FUNCTION_BLOCK Meca500_SetGripperVel
VAR
    Output_Params : array[1..6] of real;
    FirstScan : BOOL := False;
END_VAR
VAR_INPUT
    Execute : BOOL;
    Speed : REAL;
END_VAR
VAR_OUTPUT
    Sent : BOOL;
    Buffered : BOOL;
    Error : BOOL;
END_VAR
VAR_IN_OUT
    Robot : Meca500;
END_VAR
VAR_INPUT
    ExternalStateControl : BOOL;
    ExternalMoveID : UINT;
END_VAR
IF Execute THEN	
	(*Collect Inputs and store them locally*)
	Output_Params[1]:=Speed;
	Output_Params[2]:=0;
	Output_Params[3]:=0;
	Output_Params[4]:=0;
	Output_Params[5]:=0;
	Output_Params[6]:=0;

	(* If Values have change, Reinitialise Outputs*)

	IF FirstScan=0 OR 
		Robot.Outputs.MotionCommand.MoveSubIndex001 <> Output_Params[1] OR 
		Robot.Outputs.MotionCommand.MoveSubIndex002 <> Output_Params[2] OR 
		Robot.Outputs.MotionCommand.MoveSubIndex003 <> Output_Params[3] OR
		Robot.Outputs.MotionCommand.MoveSubIndex004 <> Output_Params[4] OR 
		Robot.Outputs.MotionCommand.MoveSubIndex005 <> Output_Params[5] OR 
		Robot.Outputs.MotionCommand.MoveSubIndex006 <> Output_Params[6] 
	THEN
		Buffered := FALSE;
		Sent := FALSE;
	END_IF;


	(*if not in legacy mode, Act Setpoint*)
	IF Robot.Outputs.MotionControl.MoveID <> 0 THEN
	    Robot.Outputs.MotionControl.SetPoint := TRUE;
	END_IF;

	(* To send _Move, send _Move ID *)
	IF NOT Buffered AND NOT Sent THEN
	    
	    Robot.Outputs.MotionCommand.MoveCommand	:= EnumToNum(Meca500Cmd#SetGripperVel);
	    Robot.Outputs.MotionCommand.MoveSubIndex001 := Output_Params[1];
		Robot.Outputs.MotionCommand.MoveSubIndex002 := Output_Params[2];
		Robot.Outputs.MotionCommand.MoveSubIndex003 := Output_Params[3];
		Robot.Outputs.MotionCommand.MoveSubIndex004 := Output_Params[4];
		Robot.Outputs.MotionCommand.MoveSubIndex005 := Output_Params[5];
		Robot.Outputs.MotionCommand.MoveSubIndex006 := Output_Params[6];
	    
	    IF ExternalStateControl THEN
	        IF ExternalMoveID <> 0 AND ExternalMoveID <> 32190 AND ExternalMoveID <> 32191 THEN
	            Robot.Outputs.MotionControl.MoveID := ExternalMoveID;
	            Sent := TRUE;
	        END_IF;
	        
	    ELSE (*Not External Control*)
	        IF Robot.Outputs.MotionControl.MoveID = 32190 THEN
	            Robot.Outputs.MotionControl.MoveID := 32191;
	        ELSIF Robot.Outputs.MotionControl.MoveID = 32191 THEN
	            Robot.Outputs.MotionControl.MoveID := 32190;
	        ELSIF Robot.Outputs.MotionControl.MoveID <> 32190 OR Robot.Outputs.MotionControl.MoveID <> 32191 THEN
	            Robot.Outputs.MotionControl.MoveID := 32190;
	        END_IF;
	        Sent := TRUE;
	    END_IF;
	END_IF;

	(* Check if command has been sent, if so, check if it was received *)
	IF Sent AND
	    Robot.Outputs.MotionCommand.MoveCommand = EnumToNum(Meca500Cmd#SetGripperVel) AND
	    Robot.Outputs.MotionCommand.MoveSubIndex001 = Output_Params[1] AND 
		Robot.Outputs.MotionCommand.MoveSubIndex002 = Output_Params[2] AND 
		Robot.Outputs.MotionCommand.MoveSubIndex003 = Output_Params[3] AND 
		Robot.Outputs.MotionCommand.MoveSubIndex004 = Output_Params[4] AND 
		Robot.Outputs.MotionCommand.MoveSubIndex005 = Output_Params[5] AND 
		Robot.Outputs.MotionCommand.MoveSubIndex006 = Output_Params[6] AND
		Robot.Inputs.Motion.MoveID = Robot.Outputs.MotionControl.MoveID 
	THEN
		 Buffered := TRUE;
	END_IF;


	(*If External _Move ID is equal to Internal, raise an error*)
	IF ExternalMoveID = 32190 OR ExternalMoveID = 32191 THEN
	    Error := TRUE;
	END_IF;

	FirstScan := TRUE;
ELSE
	FirstScan := False;
	Sent := FALSE;
	Buffered := FALSE;
END_IF;
END_FUNCTION_BLOCK

FUNCTION_BLOCK Meca500_SetJointsAcc
VAR
    Output_Params : array[1..6] of real;
    FirstScan : BOOL := False;
END_VAR
VAR_INPUT
    Execute : BOOL;
    Acceleration_Percentage : REAL;
END_VAR
VAR_OUTPUT
    Sent : BOOL;
    Buffered : BOOL;
    Error : BOOL;
END_VAR
VAR_IN_OUT
    Robot : Meca500;
END_VAR
VAR_INPUT
    ExternalStateControl : BOOL;
    ExternalMoveID : UINT;
END_VAR
IF Execute THEN	
	(*Collect Inputs and store them locally*)
	Output_Params[1]:=Acceleration_Percentage;
	Output_Params[2]:=0;
	Output_Params[3]:=0;
	Output_Params[4]:=0;
	Output_Params[5]:=0;
	Output_Params[6]:=0;

	(* If Values have change, Reinitialise Outputs*)

	IF FirstScan=0 OR 
		Robot.Outputs.MotionCommand.MoveSubIndex001 <> Output_Params[1] OR 
		Robot.Outputs.MotionCommand.MoveSubIndex002 <> Output_Params[2] OR 
		Robot.Outputs.MotionCommand.MoveSubIndex003 <> Output_Params[3] OR
		Robot.Outputs.MotionCommand.MoveSubIndex004 <> Output_Params[4] OR 
		Robot.Outputs.MotionCommand.MoveSubIndex005 <> Output_Params[5] OR 
		Robot.Outputs.MotionCommand.MoveSubIndex006 <> Output_Params[6] 
	THEN
		Buffered := FALSE;
		Sent := FALSE;
	END_IF;


	(*if not in legacy mode, Act Setpoint*)
	IF Robot.Outputs.MotionControl.MoveID <> 0 THEN
	    Robot.Outputs.MotionControl.SetPoint := TRUE;
	END_IF;

	(* To send _Move, send _Move ID *)
	IF NOT Buffered AND NOT Sent THEN
	    
	    Robot.Outputs.MotionCommand.MoveCommand	:= EnumToNum(Meca500Cmd#SetJointAcc);
	    Robot.Outputs.MotionCommand.MoveSubIndex001 := Output_Params[1];
		Robot.Outputs.MotionCommand.MoveSubIndex002 := Output_Params[2];
		Robot.Outputs.MotionCommand.MoveSubIndex003 := Output_Params[3];
		Robot.Outputs.MotionCommand.MoveSubIndex004 := Output_Params[4];
		Robot.Outputs.MotionCommand.MoveSubIndex005 := Output_Params[5];
		Robot.Outputs.MotionCommand.MoveSubIndex006 := Output_Params[6];
	    
	    IF ExternalStateControl THEN
	        IF ExternalMoveID <> 0 AND ExternalMoveID <> 32090 AND ExternalMoveID <> 32091 THEN
	            Robot.Outputs.MotionControl.MoveID := ExternalMoveID;
	            Sent := TRUE;
	        END_IF;
	        
	    ELSE (*Not External Control*)
	        IF Robot.Outputs.MotionControl.MoveID = 32090 THEN
	            Robot.Outputs.MotionControl.MoveID := 32091;
	        ELSIF Robot.Outputs.MotionControl.MoveID = 32091 THEN
	            Robot.Outputs.MotionControl.MoveID := 32090;
	        ELSIF Robot.Outputs.MotionControl.MoveID <> 32090 OR Robot.Outputs.MotionControl.MoveID <> 32091 THEN
	            Robot.Outputs.MotionControl.MoveID := 32090;
	        END_IF;
	        Sent := TRUE;
	    END_IF;
	END_IF;

	(* Check if command has been sent, if so, check if it was received *)
	IF Sent AND
	    Robot.Outputs.MotionCommand.MoveCommand = EnumToNum(Meca500Cmd#SetJointAcc) AND
	    Robot.Outputs.MotionCommand.MoveSubIndex001 = Output_Params[1] AND 
		Robot.Outputs.MotionCommand.MoveSubIndex002 = Output_Params[2] AND 
		Robot.Outputs.MotionCommand.MoveSubIndex003 = Output_Params[3] AND 
		Robot.Outputs.MotionCommand.MoveSubIndex004 = Output_Params[4] AND 
		Robot.Outputs.MotionCommand.MoveSubIndex005 = Output_Params[5] AND 
		Robot.Outputs.MotionCommand.MoveSubIndex006 = Output_Params[6] AND
		Robot.Inputs.Motion.MoveID = Robot.Outputs.MotionControl.MoveID 
	THEN
		 Buffered := TRUE;
	END_IF;


	(*If External _Move ID is equal to Internal, raise an error*)
	IF ExternalMoveID = 32090 OR ExternalMoveID = 32091 THEN
	    Error := TRUE;
	END_IF;

	FirstScan := TRUE;
ELSE
	FirstScan := False;
	Sent := FALSE;
	Buffered := FALSE;
END_IF;
END_FUNCTION_BLOCK

FUNCTION_BLOCK Meca500_SetJointsVel
VAR
    Output_Params : array[1..6] of real;
    FirstScan : BOOL := False;
END_VAR
VAR_INPUT
    Execute : BOOL;
    Velocity_Percentage : REAL;
END_VAR
VAR_OUTPUT
    Sent : BOOL;
    Buffered : BOOL;
    Error : BOOL;
END_VAR
VAR_IN_OUT
    Robot : Meca500;
END_VAR
VAR_INPUT
    ExternalStateControl : BOOL;
    ExternalMoveID : UINT;
END_VAR
IF Execute THEN	
	(*Collect Inputs and store them locally*)
	Output_Params[1]:=Velocity_Percentage;
	Output_Params[2]:=0;
	Output_Params[3]:=0;
	Output_Params[4]:=0;
	Output_Params[5]:=0;
	Output_Params[6]:=0;

	(* If Values have change, Reinitialise Outputs*)

	IF FirstScan=0 OR 
		Robot.Outputs.MotionCommand.MoveSubIndex001 <> Output_Params[1] OR 
		Robot.Outputs.MotionCommand.MoveSubIndex002 <> Output_Params[2] OR 
		Robot.Outputs.MotionCommand.MoveSubIndex003 <> Output_Params[3] OR
		Robot.Outputs.MotionCommand.MoveSubIndex004 <> Output_Params[4] OR 
		Robot.Outputs.MotionCommand.MoveSubIndex005 <> Output_Params[5] OR 
		Robot.Outputs.MotionCommand.MoveSubIndex006 <> Output_Params[6] 
	THEN
		Buffered := FALSE;
		Sent := FALSE;
	END_IF;


	(*if not in legacy mode, Act Setpoint*)
	IF Robot.Outputs.MotionControl.MoveID <> 0 THEN
	    Robot.Outputs.MotionControl.SetPoint := TRUE;
	END_IF;

	(* To send _Move, send _Move ID *)
	IF NOT Buffered AND NOT Sent THEN
	    
	    Robot.Outputs.MotionCommand.MoveCommand	:= EnumToNum(Meca500Cmd#SetJointVel);
	    Robot.Outputs.MotionCommand.MoveSubIndex001 := Output_Params[1];
		Robot.Outputs.MotionCommand.MoveSubIndex002 := Output_Params[2];
		Robot.Outputs.MotionCommand.MoveSubIndex003 := Output_Params[3];
		Robot.Outputs.MotionCommand.MoveSubIndex004 := Output_Params[4];
		Robot.Outputs.MotionCommand.MoveSubIndex005 := Output_Params[5];
		Robot.Outputs.MotionCommand.MoveSubIndex006 := Output_Params[6];
	    
	    IF ExternalStateControl THEN
	        IF ExternalMoveID <> 0 AND ExternalMoveID <> 32080 AND ExternalMoveID <> 32081 THEN
	            Robot.Outputs.MotionControl.MoveID := ExternalMoveID;
	            Sent := TRUE;
	        END_IF;
	        
	    ELSE (*Not External Control*)
	        IF Robot.Outputs.MotionControl.MoveID = 32080 THEN
	            Robot.Outputs.MotionControl.MoveID := 32081;
	        ELSIF Robot.Outputs.MotionControl.MoveID = 32081 THEN
	            Robot.Outputs.MotionControl.MoveID := 32080;
	        ELSIF Robot.Outputs.MotionControl.MoveID <> 32080 OR Robot.Outputs.MotionControl.MoveID <> 32081 THEN
	            Robot.Outputs.MotionControl.MoveID := 32080;
	        END_IF;
	        Sent := TRUE;
	    END_IF;
	END_IF;

	(* Check if command has been sent, if so, check if it was received *)
	IF Sent AND
	    Robot.Outputs.MotionCommand.MoveCommand = EnumToNum(Meca500Cmd#SetJointVel) AND
	    Robot.Outputs.MotionCommand.MoveSubIndex001 = Output_Params[1] AND 
		Robot.Outputs.MotionCommand.MoveSubIndex002 = Output_Params[2] AND 
		Robot.Outputs.MotionCommand.MoveSubIndex003 = Output_Params[3] AND 
		Robot.Outputs.MotionCommand.MoveSubIndex004 = Output_Params[4] AND 
		Robot.Outputs.MotionCommand.MoveSubIndex005 = Output_Params[5] AND 
		Robot.Outputs.MotionCommand.MoveSubIndex006 = Output_Params[6] AND
		Robot.Inputs.Motion.MoveID = Robot.Outputs.MotionControl.MoveID 
	THEN
		 Buffered := TRUE;
	END_IF;


	(*If External _Move ID is equal to Internal, raise an error*)
	IF ExternalMoveID = 32080 OR ExternalMoveID = 32081 THEN
	    Error := TRUE;
	END_IF;

	FirstScan := TRUE;
ELSE
	FirstScan := False;
	Sent := FALSE;
	Buffered := FALSE;
END_IF;
END_FUNCTION_BLOCK

FUNCTION_BLOCK Meca500_SetTorqueLimitCfg
VAR
    Output_Params : array[1..6] of real;
    FirstScan : BOOL := False;
END_VAR
VAR_INPUT
    Execute : BOOL;
    Severity : REAL;
    Mode : REAL;
END_VAR
VAR_OUTPUT
    Sent : BOOL;
    Buffered : BOOL;
    Error : BOOL;
END_VAR
VAR_IN_OUT
    Robot : Meca500;
END_VAR
VAR_INPUT
    ExternalStateControl : BOOL;
    ExternalMoveID : UINT;
END_VAR
IF Execute THEN	
	(*Collect Inputs and store them locally*)
	Output_Params[1]:=Severity;
	Output_Params[2]:=Mode;
	Output_Params[3]:=0;
	Output_Params[4]:=0;
	Output_Params[5]:=0;
	Output_Params[6]:=0;

	(* If Values have change, Reinitialise Outputs*)

	IF FirstScan=0 OR 
		Robot.Outputs.MotionCommand.MoveSubIndex001 <> Output_Params[1] OR 
		Robot.Outputs.MotionCommand.MoveSubIndex002 <> Output_Params[2] OR 
		Robot.Outputs.MotionCommand.MoveSubIndex003 <> Output_Params[3] OR
		Robot.Outputs.MotionCommand.MoveSubIndex004 <> Output_Params[4] OR 
		Robot.Outputs.MotionCommand.MoveSubIndex005 <> Output_Params[5] OR 
		Robot.Outputs.MotionCommand.MoveSubIndex006 <> Output_Params[6] 
	THEN
		Buffered := FALSE;
		Sent := FALSE;
	END_IF;


	(*if not in legacy mode, Act Setpoint*)
	IF Robot.Outputs.MotionControl.MoveID <> 0 THEN
	    Robot.Outputs.MotionControl.SetPoint := TRUE;
	END_IF;

	(* To send _Move, send _Move ID *)
	IF NOT Buffered AND NOT Sent THEN
	    
	    Robot.Outputs.MotionCommand.MoveCommand	:= EnumToNum(Meca500Cmd#SetTorquesLimitCfg);
	    Robot.Outputs.MotionCommand.MoveSubIndex001 := Output_Params[1];
		Robot.Outputs.MotionCommand.MoveSubIndex002 := Output_Params[2];
		Robot.Outputs.MotionCommand.MoveSubIndex003 := Output_Params[3];
		Robot.Outputs.MotionCommand.MoveSubIndex004 := Output_Params[4];
		Robot.Outputs.MotionCommand.MoveSubIndex005 := Output_Params[5];
		Robot.Outputs.MotionCommand.MoveSubIndex006 := Output_Params[6];
	    
	    IF ExternalStateControl THEN
	        IF ExternalMoveID <> 0 AND ExternalMoveID <> 32280 AND ExternalMoveID <> 32281 THEN
	            Robot.Outputs.MotionControl.MoveID := ExternalMoveID;
	            Sent := TRUE;
	        END_IF;
	        
	    ELSE (*Not External Control*)
	        IF Robot.Outputs.MotionControl.MoveID = 32280 THEN
	            Robot.Outputs.MotionControl.MoveID := 32281;
	        ELSIF Robot.Outputs.MotionControl.MoveID = 32281 THEN
	            Robot.Outputs.MotionControl.MoveID := 32280;
	        ELSIF Robot.Outputs.MotionControl.MoveID <> 32280 OR Robot.Outputs.MotionControl.MoveID <> 32281 THEN
	            Robot.Outputs.MotionControl.MoveID := 32280;
	        END_IF;
	        Sent := TRUE;
	    END_IF;
	END_IF;

	(* Check if command has been sent, if so, check if it was received *)
	IF Sent AND
	    Robot.Outputs.MotionCommand.MoveCommand = EnumToNum(Meca500Cmd#SetTorquesLimitCfg) AND
	    Robot.Outputs.MotionCommand.MoveSubIndex001 = Output_Params[1] AND 
		Robot.Outputs.MotionCommand.MoveSubIndex002 = Output_Params[2] AND 
		Robot.Outputs.MotionCommand.MoveSubIndex003 = Output_Params[3] AND 
		Robot.Outputs.MotionCommand.MoveSubIndex004 = Output_Params[4] AND 
		Robot.Outputs.MotionCommand.MoveSubIndex005 = Output_Params[5] AND 
		Robot.Outputs.MotionCommand.MoveSubIndex006 = Output_Params[6] AND
		Robot.Inputs.Motion.MoveID = Robot.Outputs.MotionControl.MoveID 
	THEN
		 Buffered := TRUE;
	END_IF;


	(*If External _Move ID is equal to Internal, raise an error*)
	IF ExternalMoveID = 32280 OR ExternalMoveID = 32281 THEN
	    Error := TRUE;
	END_IF;

	FirstScan := TRUE;
ELSE
	FirstScan := False;
	Sent := FALSE;
	Buffered := FALSE;
END_IF;
END_FUNCTION_BLOCK

FUNCTION_BLOCK Meca500_SetTorqueLimits
VAR
    Output_Params : array[1..6] of real;
    FirstScan : BOOL := False;
END_VAR
VAR_INPUT
    Execute : BOOL;
    Joint_1_Limit : REAL;
    Joint_2_Limit : REAL;
    Joint_3_Limit : REAL;
    Joint_4_Limit : REAL;
    Joint_5_Limit : REAL;
    Joint_6_Limit : REAL;
END_VAR
VAR_OUTPUT
    Sent : BOOL;
    Buffered : BOOL;
    Error : BOOL;
END_VAR
VAR_IN_OUT
    Robot : Meca500;
END_VAR
VAR_INPUT
    ExternalStateControl : BOOL;
    ExternalMoveID : UINT;
END_VAR
IF Execute THEN	
	(*Collect Inputs and store them locally*)
	Output_Params[1]:=Joint_1_Limit;
	Output_Params[2]:=Joint_2_Limit;
	Output_Params[3]:=Joint_3_Limit;
	Output_Params[4]:=Joint_4_Limit;
	Output_Params[5]:=Joint_5_Limit;
	Output_Params[6]:=Joint_6_Limit;


	(* If Values have change, Reinitialise Outputs*)

	IF FirstScan=0 OR 
		Robot.Outputs.MotionCommand.MoveSubIndex001 <> Output_Params[1] OR 
		Robot.Outputs.MotionCommand.MoveSubIndex002 <> Output_Params[2] OR 
		Robot.Outputs.MotionCommand.MoveSubIndex003 <> Output_Params[3] OR
		Robot.Outputs.MotionCommand.MoveSubIndex004 <> Output_Params[4] OR 
		Robot.Outputs.MotionCommand.MoveSubIndex005 <> Output_Params[5] OR 
		Robot.Outputs.MotionCommand.MoveSubIndex006 <> Output_Params[6] 
	THEN
		Buffered := FALSE;
		Sent := FALSE;
	END_IF;


	(*if not in legacy mode, Act Setpoint*)
	IF Robot.Outputs.MotionControl.MoveID <> 0 THEN
	    Robot.Outputs.MotionControl.SetPoint := TRUE;
	END_IF;

	(* To send _Move, send _Move ID *)
	IF NOT Buffered AND NOT Sent THEN
	    
	    Robot.Outputs.MotionCommand.MoveCommand	:= EnumToNum(Meca500Cmd#SetTorqueLimits);
	    Robot.Outputs.MotionCommand.MoveSubIndex001 := Output_Params[1];
		Robot.Outputs.MotionCommand.MoveSubIndex002 := Output_Params[2];
		Robot.Outputs.MotionCommand.MoveSubIndex003 := Output_Params[3];
		Robot.Outputs.MotionCommand.MoveSubIndex004 := Output_Params[4];
		Robot.Outputs.MotionCommand.MoveSubIndex005 := Output_Params[5];
		Robot.Outputs.MotionCommand.MoveSubIndex006 := Output_Params[6];
	    
	    IF ExternalStateControl THEN
	        IF ExternalMoveID <> 0 AND ExternalMoveID <> 32270 AND ExternalMoveID <> 32271 THEN
	            Robot.Outputs.MotionControl.MoveID := ExternalMoveID;
	            Sent := TRUE;
	        END_IF;
	        
	    ELSE (*Not External Control*)
	        IF Robot.Outputs.MotionControl.MoveID = 32270 THEN
	            Robot.Outputs.MotionControl.MoveID := 32271;
	        ELSIF Robot.Outputs.MotionControl.MoveID = 32271 THEN
	            Robot.Outputs.MotionControl.MoveID := 32270;
	        ELSIF Robot.Outputs.MotionControl.MoveID <> 32270 OR Robot.Outputs.MotionControl.MoveID <> 32271 THEN
	            Robot.Outputs.MotionControl.MoveID := 32270;
	        END_IF;
	        Sent := TRUE;
	    END_IF;
	END_IF;

	(* Check if command has been sent, if so, check if it was received *)
	IF Sent AND
	    Robot.Outputs.MotionCommand.MoveCommand = EnumToNum(Meca500Cmd#SetTorqueLimits) AND
	    Robot.Outputs.MotionCommand.MoveSubIndex001 = Output_Params[1] AND 
		Robot.Outputs.MotionCommand.MoveSubIndex002 = Output_Params[2] AND 
		Robot.Outputs.MotionCommand.MoveSubIndex003 = Output_Params[3] AND 
		Robot.Outputs.MotionCommand.MoveSubIndex004 = Output_Params[4] AND 
		Robot.Outputs.MotionCommand.MoveSubIndex005 = Output_Params[5] AND 
		Robot.Outputs.MotionCommand.MoveSubIndex006 = Output_Params[6] AND
		Robot.Inputs.Motion.MoveID = Robot.Outputs.MotionControl.MoveID 
	THEN
		 Buffered := TRUE;
	END_IF;


	(*If External _Move ID is equal to Internal, raise an error*)
	IF ExternalMoveID = 32270 OR ExternalMoveID = 32271 THEN
	    Error := TRUE;
	END_IF;

	FirstScan := TRUE;
ELSE
	FirstScan := False;
	Sent := FALSE;
	Buffered := FALSE;
END_IF;
END_FUNCTION_BLOCK

FUNCTION_BLOCK Meca500_SetTrf
VAR
    Output_Params : array[1..6] of real;
    FirstScan : BOOL := False;
END_VAR
VAR_INPUT
    Execute : BOOL;
    Pose_X_Pos : REAL;
    Pose_Y_Pos : REAL;
    Pose_Z_Pos : REAL;
    Pose_rX_Angle : REAL;
    Pose_rY_Angle : REAL;
    Pose_rZ_Angle : REAL;
END_VAR
VAR_OUTPUT
    Sent : BOOL;
    Buffered : BOOL;
    Error : BOOL;
END_VAR
VAR_IN_OUT
    Robot : Meca500;
END_VAR
VAR_INPUT
    ExternalStateControl : BOOL;
    ExternalMoveID : UINT;
END_VAR
IF Execute THEN	
	(*Collect Inputs and store them locally*)
	Output_Params[1]:=Pose_X_Pos;
	Output_Params[2]:=Pose_Y_Pos;
	Output_Params[3]:=Pose_Z_Pos;
	Output_Params[4]:=Pose_rX_Angle;
	Output_Params[5]:=Pose_rY_Angle;
	Output_Params[6]:=Pose_rZ_Angle;

	(* If Values have change, Reinitialise Outputs*)

	IF FirstScan=0 OR 
		Robot.Outputs.MotionCommand.MoveSubIndex001 <> Output_Params[1] OR 
		Robot.Outputs.MotionCommand.MoveSubIndex002 <> Output_Params[2] OR 
		Robot.Outputs.MotionCommand.MoveSubIndex003 <> Output_Params[3] OR
		Robot.Outputs.MotionCommand.MoveSubIndex004 <> Output_Params[4] OR 
		Robot.Outputs.MotionCommand.MoveSubIndex005 <> Output_Params[5] OR 
		Robot.Outputs.MotionCommand.MoveSubIndex006 <> Output_Params[6] 
	THEN
		Buffered := FALSE;
		Sent := FALSE;
	END_IF;


	(*if not in legacy mode, Act Setpoint*)
	IF Robot.Outputs.MotionControl.MoveID <> 0 THEN
	    Robot.Outputs.MotionControl.SetPoint := TRUE;
	END_IF;

	(* To send _Move, send _Move ID *)
	IF NOT Buffered AND NOT Sent THEN
	    
	    Robot.Outputs.MotionCommand.MoveCommand	:= EnumToNum(Meca500Cmd#SetTrf);
	    Robot.Outputs.MotionCommand.MoveSubIndex001 := Output_Params[1];
		Robot.Outputs.MotionCommand.MoveSubIndex002 := Output_Params[2];
		Robot.Outputs.MotionCommand.MoveSubIndex003 := Output_Params[3];
		Robot.Outputs.MotionCommand.MoveSubIndex004 := Output_Params[4];
		Robot.Outputs.MotionCommand.MoveSubIndex005 := Output_Params[5];
		Robot.Outputs.MotionCommand.MoveSubIndex006 := Output_Params[6];
	    
	    IF ExternalStateControl THEN
	        IF ExternalMoveID <> 0 AND ExternalMoveID <> 32130 AND ExternalMoveID <> 32131 THEN
	            Robot.Outputs.MotionControl.MoveID := ExternalMoveID;
	            Sent := TRUE;
	        END_IF;
	        
	    ELSE (*Not External Control*)
	        IF Robot.Outputs.MotionControl.MoveID = 32130 THEN
	            Robot.Outputs.MotionControl.MoveID := 32131;
	        ELSIF Robot.Outputs.MotionControl.MoveID = 32131 THEN
	            Robot.Outputs.MotionControl.MoveID := 32130;
	        ELSIF Robot.Outputs.MotionControl.MoveID <> 32130 OR Robot.Outputs.MotionControl.MoveID <> 32131 THEN
	            Robot.Outputs.MotionControl.MoveID := 32130;
	        END_IF;
	        Sent := TRUE;
	    END_IF;
	END_IF;

	(* Check if command has been sent, if so, check if it was received *)
	IF Sent AND
	    Robot.Outputs.MotionCommand.MoveCommand = EnumToNum(Meca500Cmd#SetTrf) AND
	    Robot.Outputs.MotionCommand.MoveSubIndex001 = Output_Params[1] AND 
		Robot.Outputs.MotionCommand.MoveSubIndex002 = Output_Params[2] AND 
		Robot.Outputs.MotionCommand.MoveSubIndex003 = Output_Params[3] AND 
		Robot.Outputs.MotionCommand.MoveSubIndex004 = Output_Params[4] AND 
		Robot.Outputs.MotionCommand.MoveSubIndex005 = Output_Params[5] AND 
		Robot.Outputs.MotionCommand.MoveSubIndex006 = Output_Params[6] AND
		Robot.Inputs.Motion.MoveID = Robot.Outputs.MotionControl.MoveID 
	THEN
		 Buffered := TRUE;
	END_IF;


	(*If External _Move ID is equal to Internal, raise an error*)
	IF ExternalMoveID = 32130 OR ExternalMoveID = 32131 THEN
	    Error := TRUE;
	END_IF;

	FirstScan := TRUE;
ELSE
	FirstScan := False;
	Sent := FALSE;
	Buffered := FALSE;
END_IF;
END_FUNCTION_BLOCK

FUNCTION_BLOCK Meca500_SetValveState
VAR
    Output_Params : array[1..6] of real;
    FirstScan : BOOL := False;
END_VAR
VAR_INPUT
    Execute : BOOL;
    V1 : REAL;
    V2 : REAL;
END_VAR
VAR_OUTPUT
    Sent : BOOL;
    Buffered : BOOL;
    Error : BOOL;
END_VAR
VAR_IN_OUT
    Robot : Meca500;
END_VAR
VAR_INPUT
    ExternalStateControl : BOOL;
    ExternalMoveID : UINT;
END_VAR
IF Execute THEN	
	(*Collect Inputs and store them locally*)
	Output_Params[1]:=V1;
	Output_Params[2]:=V2;
	Output_Params[3]:=0;
	Output_Params[4]:=0;
	Output_Params[5]:=0;
	Output_Params[6]:=0;

	(* If Values have change, Reinitialise Outputs*)

	IF FirstScan=0 OR 
		Robot.Outputs.MotionCommand.MoveSubIndex001 <> Output_Params[1] OR 
		Robot.Outputs.MotionCommand.MoveSubIndex002 <> Output_Params[2] OR 
		Robot.Outputs.MotionCommand.MoveSubIndex003 <> Output_Params[3] OR
		Robot.Outputs.MotionCommand.MoveSubIndex004 <> Output_Params[4] OR 
		Robot.Outputs.MotionCommand.MoveSubIndex005 <> Output_Params[5] OR 
		Robot.Outputs.MotionCommand.MoveSubIndex006 <> Output_Params[6] 
	THEN
		Buffered := FALSE;
		Sent := FALSE;
	END_IF;


	(*if not in legacy mode, Act Setpoint*)
	IF Robot.Outputs.MotionControl.MoveID <> 0 THEN
	    Robot.Outputs.MotionControl.SetPoint := TRUE;
	END_IF;

	(* To send _Move, send _Move ID *)
	IF NOT Buffered AND NOT Sent THEN
	    
	    Robot.Outputs.MotionCommand.MoveCommand	:= EnumToNum(Meca500Cmd#SetValveState);
	    Robot.Outputs.MotionCommand.MoveSubIndex001 := Output_Params[1];
		Robot.Outputs.MotionCommand.MoveSubIndex002 := Output_Params[2];
		Robot.Outputs.MotionCommand.MoveSubIndex003 := Output_Params[3];
		Robot.Outputs.MotionCommand.MoveSubIndex004 := Output_Params[4];
		Robot.Outputs.MotionCommand.MoveSubIndex005 := Output_Params[5];
		Robot.Outputs.MotionCommand.MoveSubIndex006 := Output_Params[6];
	    
	    IF ExternalStateControl THEN
	        IF ExternalMoveID <> 0 AND ExternalMoveID <> 32300 AND ExternalMoveID <> 32301 THEN
	            Robot.Outputs.MotionControl.MoveID := ExternalMoveID;
	            Sent := TRUE;
	        END_IF;
	        
	    ELSE (*Not External Control*)
	        IF Robot.Outputs.MotionControl.MoveID = 32300 THEN
	            Robot.Outputs.MotionControl.MoveID := 32301;
	        ELSIF Robot.Outputs.MotionControl.MoveID = 32301 THEN
	            Robot.Outputs.MotionControl.MoveID := 32300;
	        ELSIF Robot.Outputs.MotionControl.MoveID <> 32300 OR Robot.Outputs.MotionControl.MoveID <> 32301 THEN
	            Robot.Outputs.MotionControl.MoveID := 32300;
	        END_IF;
	        Sent := TRUE;
	    END_IF;
	END_IF;

	(* Check if command has been sent, if so, check if it was received *)
	IF Sent AND
	    Robot.Outputs.MotionCommand.MoveCommand = EnumToNum(Meca500Cmd#SetValveState) AND
	    Robot.Outputs.MotionCommand.MoveSubIndex001 = Output_Params[1] AND 
		Robot.Outputs.MotionCommand.MoveSubIndex002 = Output_Params[2] AND 
		Robot.Outputs.MotionCommand.MoveSubIndex003 = Output_Params[3] AND 
		Robot.Outputs.MotionCommand.MoveSubIndex004 = Output_Params[4] AND 
		Robot.Outputs.MotionCommand.MoveSubIndex005 = Output_Params[5] AND 
		Robot.Outputs.MotionCommand.MoveSubIndex006 = Output_Params[6] AND
		Robot.Inputs.Motion.MoveID = Robot.Outputs.MotionControl.MoveID 
	THEN
		 Buffered := TRUE;
	END_IF;


	(*If External _Move ID is equal to Internal, raise an error*)
	IF ExternalMoveID = 32300 OR ExternalMoveID = 32301 THEN
	    Error := TRUE;
	END_IF;

	FirstScan := TRUE;
ELSE
	FirstScan := False;
	Sent := FALSE;
	Buffered := FALSE;
END_IF;
END_FUNCTION_BLOCK

FUNCTION_BLOCK Meca500_SetVelTimeout
VAR
    Output_Params : array[1..6] of real;
    FirstScan : BOOL := False;
END_VAR
VAR_INPUT
    Execute : BOOL;
    Seconds : REAL;
END_VAR
VAR_OUTPUT
    Sent : BOOL;
    Buffered : BOOL;
    Error : BOOL;
END_VAR
VAR_IN_OUT
    Robot : Meca500;
END_VAR
VAR_INPUT
    ExternalStateControl : BOOL;
    ExternalMoveID : UINT;
END_VAR
IF Execute THEN	
	(*Collect Inputs and store them locally*)
	Output_Params[1]:=Seconds;
	Output_Params[2]:=0;
	Output_Params[3]:=0;
	Output_Params[4]:=0;
	Output_Params[5]:=0;
	Output_Params[6]:=0;


	(* If Values have change, Reinitialise Outputs*)

	IF FirstScan=0 OR 
		Robot.Outputs.MotionCommand.MoveSubIndex001 <> Output_Params[1] OR 
		Robot.Outputs.MotionCommand.MoveSubIndex002 <> Output_Params[2] OR 
		Robot.Outputs.MotionCommand.MoveSubIndex003 <> Output_Params[3] OR
		Robot.Outputs.MotionCommand.MoveSubIndex004 <> Output_Params[4] OR 
		Robot.Outputs.MotionCommand.MoveSubIndex005 <> Output_Params[5] OR 
		Robot.Outputs.MotionCommand.MoveSubIndex006 <> Output_Params[6] 
	THEN
		Buffered := FALSE;
		Sent := FALSE;
	END_IF;


	(*if not in legacy mode, Act Setpoint*)
	IF Robot.Outputs.MotionControl.MoveID <> 0 THEN
	    Robot.Outputs.MotionControl.SetPoint := TRUE;
	END_IF;

	(* To send _Move, send _Move ID *)
	IF NOT Buffered AND NOT Sent THEN
	    
	    Robot.Outputs.MotionCommand.MoveCommand	:= EnumToNum(Meca500Cmd#SetVelTimeout);
	    Robot.Outputs.MotionCommand.MoveSubIndex001 := Output_Params[1];
		Robot.Outputs.MotionCommand.MoveSubIndex002 := Output_Params[2];
		Robot.Outputs.MotionCommand.MoveSubIndex003 := Output_Params[3];
		Robot.Outputs.MotionCommand.MoveSubIndex004 := Output_Params[4];
		Robot.Outputs.MotionCommand.MoveSubIndex005 := Output_Params[5];
		Robot.Outputs.MotionCommand.MoveSubIndex006 := Output_Params[6];
	    
	    IF ExternalStateControl THEN
	        IF ExternalMoveID <> 0 AND ExternalMoveID <> 32240 AND ExternalMoveID <> 32241 THEN
	            Robot.Outputs.MotionControl.MoveID := ExternalMoveID;
	            Sent := TRUE;
	        END_IF;
	        
	    ELSE (*Not External Control*)
	        IF Robot.Outputs.MotionControl.MoveID = 32240 THEN
	            Robot.Outputs.MotionControl.MoveID := 32241;
	        ELSIF Robot.Outputs.MotionControl.MoveID = 32241 THEN
	            Robot.Outputs.MotionControl.MoveID := 32240;
	        ELSIF Robot.Outputs.MotionControl.MoveID <> 32240 OR Robot.Outputs.MotionControl.MoveID <> 32241 THEN
	            Robot.Outputs.MotionControl.MoveID := 32240;
	        END_IF;
	        Sent := TRUE;
	    END_IF;
	END_IF;

	(* Check if command has been sent, if so, check if it was received *)
	IF Sent AND
	    Robot.Outputs.MotionCommand.MoveCommand = EnumToNum(Meca500Cmd#SetVelTimeout) AND
	    Robot.Outputs.MotionCommand.MoveSubIndex001 = Output_Params[1] AND 
		Robot.Outputs.MotionCommand.MoveSubIndex002 = Output_Params[2] AND 
		Robot.Outputs.MotionCommand.MoveSubIndex003 = Output_Params[3] AND 
		Robot.Outputs.MotionCommand.MoveSubIndex004 = Output_Params[4] AND 
		Robot.Outputs.MotionCommand.MoveSubIndex005 = Output_Params[5] AND 
		Robot.Outputs.MotionCommand.MoveSubIndex006 = Output_Params[6] AND
		Robot.Inputs.Motion.MoveID = Robot.Outputs.MotionControl.MoveID 
	THEN
		 Buffered := TRUE;
	END_IF;


	(*If External _Move ID is equal to Internal, raise an error*)
	IF ExternalMoveID = 32240 OR ExternalMoveID = 32241 THEN
	    Error := TRUE;
	END_IF;

	FirstScan := TRUE;
ELSE
	FirstScan := False;
	Sent := FALSE;
	Buffered := FALSE;
END_IF;
END_FUNCTION_BLOCK

FUNCTION_BLOCK Meca500_SetWrf
VAR
    Output_Params : array[1..6] of real;
    FirstScan : BOOL := False;
END_VAR
VAR_INPUT
    Execute : BOOL;
    Pose_X_Pos : REAL;
    Pose_Y_Pos : REAL;
    Pose_Z_Pos : REAL;
    Pose_rX_Angle : REAL;
    Pose_rY_Angle : REAL;
    Pose_rZ_Angle : REAL;
END_VAR
VAR_OUTPUT
    Sent : BOOL;
    Buffered : BOOL;
    Error : BOOL;
END_VAR
VAR_IN_OUT
    Robot : Meca500;
END_VAR
VAR_INPUT
    ExternalStateControl : BOOL;
    ExternalMoveID : UINT;
END_VAR
IF Execute THEN	
	(*Collect Inputs and store them locally*)
	Output_Params[1]:=Pose_X_Pos;
	Output_Params[2]:=Pose_Y_Pos;
	Output_Params[3]:=Pose_Z_Pos;
	Output_Params[4]:=Pose_rX_Angle;
	Output_Params[5]:=Pose_rY_Angle;
	Output_Params[6]:=Pose_rZ_Angle;

	(* If Values have change, Reinitialise Outputs*)

	IF FirstScan=0 OR 
		Robot.Outputs.MotionCommand.MoveSubIndex001 <> Output_Params[1] OR 
		Robot.Outputs.MotionCommand.MoveSubIndex002 <> Output_Params[2] OR 
		Robot.Outputs.MotionCommand.MoveSubIndex003 <> Output_Params[3] OR
		Robot.Outputs.MotionCommand.MoveSubIndex004 <> Output_Params[4] OR 
		Robot.Outputs.MotionCommand.MoveSubIndex005 <> Output_Params[5] OR 
		Robot.Outputs.MotionCommand.MoveSubIndex006 <> Output_Params[6] 
	THEN
		Buffered := FALSE;
		Sent := FALSE;
	END_IF;


	(*if not in legacy mode, Act Setpoint*)
	IF Robot.Outputs.MotionControl.MoveID <> 0 THEN
	    Robot.Outputs.MotionControl.SetPoint := TRUE;
	END_IF;

	(* To send _Move, send _Move ID *)
	IF NOT Buffered AND NOT Sent THEN
	    
	    Robot.Outputs.MotionCommand.MoveCommand	:= EnumToNum(Meca500Cmd#SetWrf);
	    Robot.Outputs.MotionCommand.MoveSubIndex001 := Output_Params[1];
		Robot.Outputs.MotionCommand.MoveSubIndex002 := Output_Params[2];
		Robot.Outputs.MotionCommand.MoveSubIndex003 := Output_Params[3];
		Robot.Outputs.MotionCommand.MoveSubIndex004 := Output_Params[4];
		Robot.Outputs.MotionCommand.MoveSubIndex005 := Output_Params[5];
		Robot.Outputs.MotionCommand.MoveSubIndex006 := Output_Params[6];
	    
	    IF ExternalStateControl THEN
	        IF ExternalMoveID <> 0 AND ExternalMoveID <> 32140 AND ExternalMoveID <> 32141 THEN
	            Robot.Outputs.MotionControl.MoveID := ExternalMoveID;
	            Sent := TRUE;
	        END_IF;
	        
	    ELSE (*Not External Control*)
	        IF Robot.Outputs.MotionControl.MoveID = 32140 THEN
	            Robot.Outputs.MotionControl.MoveID := 32141;
	        ELSIF Robot.Outputs.MotionControl.MoveID = 32141 THEN
	            Robot.Outputs.MotionControl.MoveID := 32140;
	        ELSIF Robot.Outputs.MotionControl.MoveID <> 32140 OR Robot.Outputs.MotionControl.MoveID <> 32141 THEN
	            Robot.Outputs.MotionControl.MoveID := 32140;
	        END_IF;
	        Sent := TRUE;
	    END_IF;
	END_IF;

	(* Check if command has been sent, if so, check if it was received *)
	IF Sent AND
	    Robot.Outputs.MotionCommand.MoveCommand = EnumToNum(Meca500Cmd#SetWrf) AND
	    Robot.Outputs.MotionCommand.MoveSubIndex001 = Output_Params[1] AND 
		Robot.Outputs.MotionCommand.MoveSubIndex002 = Output_Params[2] AND 
		Robot.Outputs.MotionCommand.MoveSubIndex003 = Output_Params[3] AND 
		Robot.Outputs.MotionCommand.MoveSubIndex004 = Output_Params[4] AND 
		Robot.Outputs.MotionCommand.MoveSubIndex005 = Output_Params[5] AND 
		Robot.Outputs.MotionCommand.MoveSubIndex006 = Output_Params[6] AND
		Robot.Inputs.Motion.MoveID = Robot.Outputs.MotionControl.MoveID 
	THEN
		 Buffered := TRUE;
	END_IF;


	(*If External _Move ID is equal to Internal, raise an error*)
	IF ExternalMoveID = 32140 OR ExternalMoveID = 32141 THEN
	    Error := TRUE;
	END_IF;

	FirstScan := TRUE;
ELSE
	FirstScan := False;
	Sent := FALSE;
	Buffered := FALSE;
END_IF;
END_FUNCTION_BLOCK

FUNCTION_BLOCK Meca500_StartProgram
VAR
    Output_Params : array[1..6] of real;
    FirstScan : BOOL := False;
END_VAR
VAR_INPUT
    Execute : BOOL;
    n : REAL;
END_VAR
VAR_OUTPUT
    Sent : BOOL;
    Buffered : BOOL;
    Error : BOOL;
END_VAR
VAR_IN_OUT
    Robot : Meca500;
END_VAR
VAR_INPUT
    ExternalStateControl : BOOL;
    ExternalMoveID : UINT;
END_VAR
IF Execute THEN	
	(*Collect Inputs and store them locally*)
	Output_Params[1]:=n;
	Output_Params[2]:=0;
	Output_Params[3]:=0;
	Output_Params[4]:=0;
	Output_Params[5]:=0;
	Output_Params[6]:=0;


	(* If Values have change, Reinitialise Outputs*)

	IF FirstScan=0 OR 
		Robot.Outputs.MotionCommand.MoveSubIndex001 <> Output_Params[1] OR 
		Robot.Outputs.MotionCommand.MoveSubIndex002 <> Output_Params[2] OR 
		Robot.Outputs.MotionCommand.MoveSubIndex003 <> Output_Params[3] OR
		Robot.Outputs.MotionCommand.MoveSubIndex004 <> Output_Params[4] OR 
		Robot.Outputs.MotionCommand.MoveSubIndex005 <> Output_Params[5] OR 
		Robot.Outputs.MotionCommand.MoveSubIndex006 <> Output_Params[6] 
	THEN
		Buffered := FALSE;
		Sent := FALSE;
	END_IF;


	(*if not in legacy mode, Act Setpoint*)
	IF Robot.Outputs.MotionControl.MoveID <> 0 THEN
	    Robot.Outputs.MotionControl.SetPoint := TRUE;
	END_IF;

	(* To send _Move, send _Move ID *)
	IF NOT Buffered AND NOT Sent THEN
	    
	    Robot.Outputs.MotionCommand.MoveCommand	:= EnumToNum(Meca500Cmd#StartProgram);
	    Robot.Outputs.MotionCommand.MoveSubIndex001 := Output_Params[1];
		Robot.Outputs.MotionCommand.MoveSubIndex002 := Output_Params[2];
		Robot.Outputs.MotionCommand.MoveSubIndex003 := Output_Params[3];
		Robot.Outputs.MotionCommand.MoveSubIndex004 := Output_Params[4];
		Robot.Outputs.MotionCommand.MoveSubIndex005 := Output_Params[5];
		Robot.Outputs.MotionCommand.MoveSubIndex006 := Output_Params[6];
	    
	    IF ExternalStateControl THEN
	        IF ExternalMoveID <> 0 AND ExternalMoveID <> 31900 AND ExternalMoveID <> 31901 THEN
	            Robot.Outputs.MotionControl.MoveID := ExternalMoveID;
	            Sent := TRUE;
	        END_IF;
	        
	    ELSE (*Not External Control*)
	        IF Robot.Outputs.MotionControl.MoveID = 31900 THEN
	            Robot.Outputs.MotionControl.MoveID := 31901;
	        ELSIF Robot.Outputs.MotionControl.MoveID = 31901 THEN
	            Robot.Outputs.MotionControl.MoveID := 31900;
	        ELSIF Robot.Outputs.MotionControl.MoveID <> 31900 OR Robot.Outputs.MotionControl.MoveID <> 31901 THEN
	            Robot.Outputs.MotionControl.MoveID := 31900;
	        END_IF;
	        Sent := TRUE;
	    END_IF;
	END_IF;

	(* Check if command has been sent, if so, check if it was received *)
	IF Sent AND
	    Robot.Outputs.MotionCommand.MoveCommand = EnumToNum(Meca500Cmd#StartProgram) AND
	    Robot.Outputs.MotionCommand.MoveSubIndex001 = Output_Params[1] AND 
		Robot.Outputs.MotionCommand.MoveSubIndex002 = Output_Params[2] AND 
		Robot.Outputs.MotionCommand.MoveSubIndex003 = Output_Params[3] AND 
		Robot.Outputs.MotionCommand.MoveSubIndex004 = Output_Params[4] AND 
		Robot.Outputs.MotionCommand.MoveSubIndex005 = Output_Params[5] AND 
		Robot.Outputs.MotionCommand.MoveSubIndex006 = Output_Params[6] AND
		Robot.Inputs.Motion.MoveID = Robot.Outputs.MotionControl.MoveID 
	THEN
		 Buffered := TRUE;
	END_IF;


	(*If External _Move ID is equal to Internal, raise an error*)
	IF ExternalMoveID = 31900 OR ExternalMoveID = 31901 THEN
	    Error := TRUE;
	END_IF;

	FirstScan := TRUE;
ELSE
	FirstScan := False;
	Sent := FALSE;
	Buffered := FALSE;
END_IF;
END_FUNCTION_BLOCK